Universal Robots PolyScope program: canpickerclient.urp

Program canpickerclient (installation=default directory=/programs/usbdisk createdIn=3.15.0.106151 lastSavedIn=3.15.0.106151 robotSerialNumber=2019300132)
Calibrated DH parameters: a=[0.000112, -0.61042, -0.561772, 0.000081, -0.000061, 0]; d=[0.12813, 3.389544, -34.235274, 31.009166, 0.115682, 0.092085]; alpha=[1.570643, -0.014365, -0.003345, 1.570403, -1.570673, 0]; deltaTheta=[-0.000108, -0.071637, 0.2557, -0.186277, 0.001922, -0.00065]
BeforeStart
  rpicon := rpc_factory("xmlrpc","http://192.168.1.100:50001")
Robot Program (runOnlyOnce=false)
  mid := Point_4
  Loop Forever
    MoveJ speed 60 deg/s, acceleration 80 deg/s^2 (useActiveTCP=true)
      URCap RG6 (RG - On Robot, OnRobot A/S) dataModel(depthCompensate=false, payload=0.0, force=50, width=20, name=RG6(20))
      Waypoint homepose: TCP in base x=503.078 y=294.269 z=399.963 mm, rx=-1.4434 ry=-2.7661 rz=0.006 rad; joints [44.97, -78.954, -101.241, -90.249, 90.928, 10.937] deg; flange x=507.966 y=292.733 z=634.257 mm, rx=2.7817 ry=-1.4515 rz=-0.0338 rad
    TinAvailable := False
    Loop While (checkContinuously=false) expression=TinAvailable== False
      TinAvailable := rpicon.requestIsEmptyTin()
    TinTopPose := rpicon.requestEmptyTinTopPose()
    MoveJ speed 60 deg/s, acceleration 80 deg/s^2 (useActiveTCP=true)
      Waypoint Waypoint (Variable): variable=TinTopPose
    URCap RG6 (RG - On Robot, OnRobot A/S) dataModel(depthCompensate=false, force=120, payload=0.0, width=120, name=RG6(120))
    JointAngles := rpicon.requestGripperRotationJointAngles(get_target_joint_positions(), 0)
    RotatedPose := get_forward_kin(JointAngles)
    MoveJ speed 60 deg/s, acceleration 80 deg/s^2 (useActiveTCP=true)
      Waypoint Waypoint (Variable): variable=RotatedPose
    TinScanPose := rpicon.requestEmptyTinScanPose(RotatedPose)
    MoveL speed 250 mm/s, acceleration 1200 mm/s^2 (useActiveTCP=true) feature=Base
      Waypoint Waypoint (Variable): variable=TinScanPose
    RfidVal := rpicon.requestRFIDValidation()
    If RfidVal == False
      MoveL speed 250 mm/s, acceleration 1200 mm/s^2 (useActiveTCP=true) feature=Base
        Waypoint Waypoint (Variable): variable=RotatedPose
      JointAngles := rpicon.requestGripperRotationJointAngles(get_target_joint_positions(), -179)
      RotatedPose := get_forward_kin(JointAngles)
      MoveJ speed 60 deg/s, acceleration 80 deg/s^2 (useActiveTCP=true)
        Waypoint Waypoint (Variable): variable=RotatedPose
      TinScanPose := rpicon.requestEmptyTinScanPose(RotatedPose)
      MoveL speed 250 mm/s, acceleration 1200 mm/s^2 (useActiveTCP=true) feature=Base
        Waypoint Waypoint (Variable): variable=TinScanPose
      Wait Sleep waitTime=3
      TinGrabPose := rpicon.requestEmptyTinGrabPose(RotatedPose)
      MoveL speed 250 mm/s, acceleration 1200 mm/s^2 (useActiveTCP=true) feature=Base
        Waypoint Waypoint (Variable): variable=TinGrabPose
      Wait Sleep waitTime=3
    TinGrabPose := rpicon.requestEmptyTinGrabPose(RotatedPose)
    MoveL speed 250 mm/s, acceleration 1200 mm/s^2 (useActiveTCP=true) feature=Base
      Waypoint Waypoint (Variable): variable=TinGrabPose
    Wait Sleep waitTime=3
    URCap RG6 (RG - On Robot, OnRobot A/S) dataModel(depthCompensate=false, payload=0.0, force=50, width=50, name=RG6(50))
    TinLeavePose := rpicon.requestEmptyTinLeavePose(TinGrabPose)
    MoveL speed 250 mm/s, acceleration 1200 mm/s^2 (useActiveTCP=true) feature=Base
      Waypoint Waypoint (Variable): variable=TinLeavePose
    If RfidVal== True
      MoveJ speed 60 deg/s, acceleration 80 deg/s^2 (useActiveTCP=true)
        Waypoint Waypoint (Variable): variable=mid
      CaningTopPose := rpicon.requestCaningTopPose()
      MoveJ speed 60 deg/s, acceleration 80 deg/s^2 (useActiveTCP=true)
        Waypoint Waypoint (Variable): variable=CaningTopPose
      CaningGrabPose := rpicon.requestCaningGrabPose(CaningTopPose)
      MoveL speed 250 mm/s, acceleration 1200 mm/s^2 (useActiveTCP=true) feature=Base
        Waypoint Waypoint (Variable): variable=CaningGrabPose
      URCap RG6 (RG - On Robot, OnRobot A/S) dataModel(depthCompensate=false, payload=0.0, width=120, force=50, name=RG6(120))
      MoveL speed 250 mm/s, acceleration 1200 mm/s^2 (useActiveTCP=true) feature=Base
        Waypoint Waypoint (Variable): variable=CaningTopPose
      Wait Sleep waitTime=3
      sealhome := Point_5
      MoveL speed 250 mm/s, acceleration 1200 mm/s^2 (useActiveTCP=true) feature=Base
        Waypoint Waypoint (Variable): variable=sealhome
        Wait Sleep waitTime=3
        Wait Sleep waitTime=3
      SealVal := rpicon.requestSealValidation()
      SuppressedNode
        MoveL speed 250 mm/s, acceleration 1200 mm/s^2 (useActiveTCP=true) feature=Base
          Waypoint Waypoint (Variable): variable=CaningTopPose
      MoveJ speed 60 deg/s, acceleration 80 deg/s^2 (useActiveTCP=true)
        Waypoint Waypoint (Variable): variable=CaningGrabPose
      Wait Sleep waitTime=3
      CaningScanPose := rpicon.requestCaningScanPose(CaningGrabPose)
      MoveL speed 250 mm/s, acceleration 1200 mm/s^2 (useActiveTCP=true) feature=Base
        Waypoint Waypoint (Variable): variable=CaningScanPose
      Wait Sleep waitTime=3
      RfidUpdate := rpicon.requestIsTinUpdated(SealVal)
      Wait Sleep waitTime=3
      MoveL speed 250 mm/s, acceleration 1200 mm/s^2 (useActiveTCP=true) feature=Base
        Waypoint Waypoint (Variable): variable=CaningGrabPose
      Wait Sleep waitTime=3
      URCap RG6 (RG - On Robot, OnRobot A/S) dataModel(depthCompensate=false, payload=0.0, force=50, width=50, name=RG6(50))
      MoveL speed 250 mm/s, acceleration 1200 mm/s^2 (useActiveTCP=true) feature=Base
        Waypoint Waypoint (Variable): variable=CaningTopPose
      If SealVal== True  and  RfidUpdate== True
        pvTopNextPose := rpicon.requestPackingValidTopNextPose()
        MoveJ speed 60 deg/s, acceleration 80 deg/s^2 (useActiveTCP=true)
          Waypoint Waypoint (Variable): variable=pvTopNextPose
        pvRelNextPose := rpicon.requestPackingValidReleaseNextPose(pvTopNextPose)
        MoveL speed 250 mm/s, acceleration 1200 mm/s^2 (useActiveTCP=true) feature=Base
          Waypoint Waypoint (Variable): variable=pvRelNextPose
        URCap RG6 (RG - On Robot, OnRobot A/S) dataModel(depthCompensate=false, payload=0.0, width=120, force=50, name=RG6(120))
        MoveL speed 250 mm/s, acceleration 1200 mm/s^2 (useActiveTCP=true) feature=Base
          Waypoint Waypoint (Variable): variable=pvTopNextPose
      Else 
        pnvTopNextPose := rpicon.requestPackingNotValidTopNextPose()
        MoveJ speed 60 deg/s, acceleration 80 deg/s^2 (useActiveTCP=true)
          Waypoint Waypoint (Variable): variable=pnvTopNextPose
        pnvRelNextPose := rpicon.requestPackingNotValidReleaseNextPose(pnvTopNextPose)
        MoveL speed 250 mm/s, acceleration 1200 mm/s^2 (useActiveTCP=true) feature=Base
          Waypoint Waypoint (Variable): variable=pnvRelNextPose
        URCap RG6 (RG - On Robot, OnRobot A/S) dataModel(depthCompensate=false, payload=0.0, width=120, force=50, name=RG6(120))
        MoveL speed 250 mm/s, acceleration 1200 mm/s^2 (useActiveTCP=true) feature=Base
          Waypoint Waypoint (Variable): variable=pnvTopNextPose
    Else 
      CaningTopPose := rpicon.requestCaningTopPose()
      MoveJ speed 60 deg/s, acceleration 80 deg/s^2 (useActiveTCP=true)
        Waypoint Waypoint (Variable): variable=mid
      MoveJ speed 60 deg/s, acceleration 80 deg/s^2 (useActiveTCP=true)
        Waypoint Waypoint (Variable): variable=CaningTopPose
      pnvTopNextPose := rpicon.requestPackingNotValidTopNextPose()
      MoveJ speed 60 deg/s, acceleration 80 deg/s^2 (useActiveTCP=true)
        Waypoint Waypoint (Variable): variable=pnvTopNextPose
      pnvRelNextPose := rpicon.requestPackingNotValidReleaseNextPose(pnvTopNextPose)
      MoveL speed 250 mm/s, acceleration 1200 mm/s^2 (useActiveTCP=true) feature=Base
        Waypoint Waypoint (Variable): variable=pnvRelNextPose
      Wait Sleep waitTime=3
      URCap RG6 (RG - On Robot, OnRobot A/S) dataModel(depthCompensate=false, payload=0.0, width=120, force=50, name=RG6(120))
      MoveL speed 250 mm/s, acceleration 1200 mm/s^2 (useActiveTCP=true) feature=Base
        Waypoint Waypoint (Variable): variable=pnvTopNextPose
